(* CODESYS project TP_INF_IND_RENAN_JULIA.project

Project tree, tasks and I/O mapping:
  Device : CODESYS Control Win V3, 3S - Smart Software Solutions GmbH, order no. 305021, version 3.5.11.40
    application Application
      libraries: Standard, * (System)
      task MainTask (cyclic, interval t#10ms, priority 1) calls Main
      task SimulacaoTask (cyclic, interval t#100ms, priority 1) calls SimulacaoProcesso
      program Main [ST]
      program SimulacaoProcesso [ST]
      global variables Variaveis_globais
      function block ControleCarregamento [ST]
      function block ControleDescarregamento [ST]
      function block ManualControl [ST]
      function block gestaoAlarmes [ST]
*)

// Device/Application/Variaveis_globais

VAR_GLOBAL
    // Variáveis de Peso dos Silos
    PESO_SILO1: REAL;
    PESO_SILO2: REAL;
	PESO_MOEGA: REAL;
	CAPACIDADE_SILO : REAL := 2500;
	CAPACIDADE_VAGAO: INT  := 1000;
	CAPACIDADE_ARMAZENAMENTO_SILOS : REAL;
	CAMINHAO_CAPAZ : BOOL;
	INICIAR_CARREGAMENTO : BOOL;
	INICIAR_DESCARREGAMENTO : BOOL;
	VAGAO_POSICIONADO : BOOL;
	PESO_TRANSPORTADOR_ENTRADA : REAL;

    // Indicadores de Nível Alto dos Silos
    NIVEL_ALTO_SILO1: BOOL;
    NIVEL_ALTO_SILO2: BOOL;
    NIVEL_BAIXO_SILO1: BOOL;
	NIVEL_BAIXO_SILO2: BOOL;
    // Posicionamento do Caminhão
    CAMINHAO_POSICIONADO: BOOL;

    // Capacidade do Caminhão
    CAPACIDADE_CAMINHAO: REAL;

    // Comandos para Iniciar Processos
    CMD_INICIAR_DESCARREGAMENTO: BOOL;
    CMD_INICIAR_CARREGAMENTO: BOOL;

    // Estados dos Transportadores
    TRANSPORTADOR_ENTRADA_ON: BOOL;
    TRANSPORTADOR_SAIDA_ON: BOOL;

    // Estados de Ventilação dos Silos
    VENTILACAO_SILO1: BOOL;
    VENTILACAO_SILO2: BOOL;

    // Estado do Alimentador da Moega
    ALIMENTADOR_MOEGA1_ON: BOOL;
	ALIMENTADOR_MOEGA2_ON: BOOL;
	SENSOR_ALIMENTADOR_MOEGA1: BOOL;
	SENSOR_ALIMENTADOR_MOEGA2: BOOL;
    
    // Estados dos Alimentadores de Saída
    ALIMENTADOR_SAIDA_ON: BOOL;
    MOEGA_PESAGEM_ON: BOOL;
    ALIMENTADOR_MOEGA1: BOOL;
    ALIMENTADOR_MOEGA2: BOOL;
	

    // Posição do Desviador de Mangueira
    DESVIADOR_MANGUEIRA_POS: INT;

    // Alarmes
    ALARME_ALIMENTADOR_SAIDA: BOOL;
    ALARME_TRANSPORTADOR_ENTRADA: BOOL;
    ALARME_TRANSPORTADOR_SAIDA: BOOL;
    ALARME_VENTILACAO_SILO1: BOOL;
    ALARME_VENTILACAO_SILO2: BOOL;
	ALARME_CARREGAMENTO: BOOL;
	ALARME_MOEGA: BOOL;
	ALARME_ALIMENTADOR_MOEGA1: BOOL;
	ALARME_ALIMENTADOR_MOEGA2: BOOL;
	ALARME_DESCARREGAMENTO : BOOL;

    // Comandos Manuais
    MANUAL_CMD_TRANSPORTADOR_ENTRADA: BOOL;
    MANUAL_CMD_TRANSPORTADOR_SAIDA: BOOL;
    MANUAL_CMD_VENTILACAO_SILO1: BOOL;
    MANUAL_CMD_VENTILACAO_SILO2: BOOL;
    MANUAL_CMD_ALIMENTADOR_MOEGA: BOOL;

    // Sensores de Posicionamento
    SENSOR_POSICIONAMENTO_VAGAO: BOOL;
    SENSOR_POSICIONAMENTO_CAMINHAO: BOOL;
END_VAR

// Device/Application/Main
PROGRAM Main
VAR
    mode: BOOL; 
    controleDescarregamento: ControleDescarregamento;
    controleCarregamento: ControleCarregamento;
   // simulacaoProcesso: SimulacaoProcesso;
    gestaoAlarmes: GestaoAlarmes;
    manualControl: ManualControl;
    
END_VAR

// Chamar os blocos de controle conforme o modo de operação
IF mode THEN // Modo automático
    controleDescarregamento();
    controleCarregamento();
ELSE // Modo manual
    manualControl();
END_IF

// Simulação e gestão de alarmes
//simulacaoProcesso();
gestaoAlarmes();

END_PROGRAM

// Device/Application/ControleDescarregamento
FUNCTION_BLOCK ControleDescarregamento
VAR
    tempo: TIME := T#0s;
    inicio_descarregamento: TIME;
END_VAR

CAPACIDADE_ARMAZENAMENTO_SILOS := (2400 - PESO_SILO1) + (2400 - PESO_SILO2);


IF (CAPACIDADE_ARMAZENAMENTO_SILOS >= CAPACIDADE_VAGAO) AND (VAGAO_POSICIONADO) THEN
	IF CMD_INICIAR_DESCARREGAMENTO THEN
		IF (NOT VENTILACAO_SILO2) AND (NOT VENTILACAO_SILO1) AND (NOT TRANSPORTADOR_ENTRADA_ON) THEN
          IF (NOT ALARME_TRANSPORTADOR_ENTRADA) AND (NOT ALARME_TRANSPORTADOR_SAIDA) AND (NOT ALARME_VENTILACAO_SILO1) AND (NOT ALARME_VENTILACAO_SILO2) AND (NOT ALARME_ALIMENTADOR_MOEGA1)AND (NOT ALARME_ALIMENTADOR_MOEGA2) AND (NOT ALARME_ALIMENTADOR_SAIDA) AND (NOT ALARME_MOEGA) THEN
		          INICIAR_DESCARREGAMENTO := TRUE;
	      ELSE
		          INICIAR_DESCARREGAMENTO := FALSE;
		          ALARME_DESCARREGAMENTO  := TRUE;
		  END_IF
		END_IF
	END_IF
ELSE
	 INICIAR_DESCARREGAMENTO := FALSE;
     ALARME_DESCARREGAMENTO  := TRUE;
END_IF


IF INICIAR_DESCARREGAMENTO THEN
	
    IF (PESO_SILO1 > PESO_SILO2) OR (PESO_SILO1 = PESO_SILO2 AND DESVIADOR_MANGUEIRA_POS = 2) THEN
        DESVIADOR_MANGUEIRA_POS := 2;
        VENTILACAO_SILO2 := TRUE;
        ALIMENTADOR_MOEGA2_ON := TRUE;
        TRANSPORTADOR_ENTRADA_ON := TRUE;
        inicio_descarregamento := TIME();

        IF (NIVEL_ALTO_SILO2) THEN
            ALIMENTADOR_MOEGA2_ON := FALSE;
            TRANSPORTADOR_ENTRADA_ON := FALSE;
            VENTILACAO_SILO2 := FALSE;
            DESVIADOR_MANGUEIRA_POS := 1;
        END_IF
		
    ELSE
        DESVIADOR_MANGUEIRA_POS := 1;
        VENTILACAO_SILO1 := TRUE;
        ALIMENTADOR_MOEGA1_ON := TRUE;
        TRANSPORTADOR_ENTRADA_ON := TRUE;
        inicio_descarregamento := TIME();

        IF (NIVEL_ALTO_SILO1) THEN
            ALIMENTADOR_MOEGA1_ON := FALSE;
            TRANSPORTADOR_ENTRADA_ON := FALSE;
            VENTILACAO_SILO1 := FALSE;
            DESVIADOR_MANGUEIRA_POS := 2;
        END_IF

    END_IF
END_IF

IF PESO_TRANSPORTADOR_ENTRADA = 0 THEN

            tempo := TIME() - inicio_descarregamento;
            IF (tempo >= T#2S) THEN
               TRANSPORTADOR_ENTRADA_ON := FALSE;
            END_IF
            IF (tempo >= T#5S) THEN
               VENTILACAO_SILO1 := FALSE;
			   VENTILACAO_SILO2 := FALSE;
            END_IF
		
END_IF

END_FUNCTION_BLOCK

// Device/Application/ControleCarregamento
FUNCTION_BLOCK ControleCarregamento
VAR
    tempo: TIME := T#0s;
    inicio_carregamento: TIME;
    INICIAR_CARREGAMENTO: BOOL := FALSE;
    ALARME_CARREGAMENTO: BOOL := FALSE;
    CAPACIDADE_CAMINHAO: REAL := 0.0; // Inicialização para um valor padrão
    CAMINHAO_CAPAZ: BOOL := FALSE;
    CAMINHAO_POSICIONADO: BOOL := FALSE;
    PESO_SILO1: REAL := 0.0; // Inicialização para um valor padrão
    PESO_SILO2: REAL := 0.0; // Inicialização para um valor padrão
    VENTILACAO_SILO1: BOOL := FALSE;
    VENTILACAO_SILO2: BOOL := FALSE;
    TRANSPORTADOR_ENTRADA_ON: BOOL := FALSE;
    SENSOR_ALIMENTADOR_MOEGA1: BOOL := FALSE;
    SENSOR_ALIMENTADOR_MOEGA2: BOOL := FALSE;
    ALIMENTADOR_SAIDA_ON: BOOL := FALSE;
    TRANSPORTADOR_SAIDA_ON: BOOL := FALSE;
    MOEGA_PESAGEM_ON: BOOL := FALSE;
    ALIMENTADOR_MOEGA1_ON: BOOL := FALSE;
    ALIMENTADOR_MOEGA2_ON: BOOL := FALSE;
    ALARME_TRANSPORTADOR_ENTRADA: BOOL := FALSE;
    ALARME_TRANSPORTADOR_SAIDA: BOOL := FALSE;
    ALARME_VENTILACAO_SILO1: BOOL := FALSE;
    ALARME_VENTILACAO_SILO2: BOOL := FALSE;
    ALARME_ALIMENTADOR_MOEGA1: BOOL := FALSE;
    ALARME_ALIMENTADOR_MOEGA2: BOOL := FALSE;
    ALARME_ALIMENTADOR_SAIDA: BOOL := FALSE;
    ALARME_MOEGA: BOOL := FALSE;
END_VAR

IF (CAPACIDADE_CAMINHAO >= 200) AND (CAPACIDADE_CAMINHAO <= 800)THEN
	CAMINHAO_CAPAZ := TRUE;
ELSE
	CAMINHAO_CAPAZ := FALSE;
END_IF

IF CAMINHAO_CAPAZ AND CAMINHAO_POSICIONADO THEN //VERIFICA SE O CAMINHAO TEM CAPACIDADE E ESTÁ POSICIONADO
	IF CMD_INICIAR_CARREGAMENTO THEN            //SE RECEBER COMANDO DO OPERADOR  
  		 IF (NOT VENTILACAO_SILO2) AND (NOT VENTILACAO_SILO1) AND (NOT TRANSPORTADOR_ENTRADA_ON) AND (NOT SENSOR_ALIMENTADOR_MOEGA1) AND (NOT SENSOR_ALIMENTADOR_MOEGA2) AND (NOT ALIMENTADOR_SAIDA_ON) AND (NOT TRANSPORTADOR_SAIDA_ON) AND (NOT MOEGA_PESAGEM_ON) AND (NOT ALIMENTADOR_MOEGA1) AND (NOT ALIMENTADOR_MOEGA2) THEN
			 IF (NOT ALARME_TRANSPORTADOR_ENTRADA) AND (NOT ALARME_TRANSPORTADOR_SAIDA) AND (NOT ALARME_VENTILACAO_SILO1) AND (NOT ALARME_VENTILACAO_SILO2) AND (NOT ALARME_ALIMENTADOR_MOEGA1)AND (NOT ALARME_ALIMENTADOR_MOEGA2) AND (NOT ALARME_ALIMENTADOR_SAIDA) AND (NOT ALARME_MOEGA) THEN
				 IF (PESO_SILO1 - 100) + (PESO_SILO2 - 100) >= CAPACIDADE_CAMINHAO THEN
                    INICIAR_CARREGAMENTO := TRUE;
                ELSE
                    ALARME_CARREGAMENTO := TRUE;
					INICIAR_CARREGAMENTO := FALSE;
                END_IF
            END_IF
        END_IF
    END_IF
END_IF

IF INICIAR_CARREGAMENTO THEN
    IF (PESO_SILO1 >= PESO_SILO2) THEN
        VENTILACAO_SILO1 := TRUE;
        ALIMENTADOR_SAIDA_ON := TRUE;
        TRANSPORTADOR_SAIDA_ON := TRUE;
        MOEGA_PESAGEM_ON := TRUE;
        ALIMENTADOR_MOEGA1 := TRUE;

        // Esperar até que a pesagem atinja o valor informado
        IF (PESO_MOEGA >= CAPACIDADE_CAMINHAO) THEN
            ALIMENTADOR_MOEGA1 := FALSE;
            VENTILACAO_SILO1 := FALSE;
            ALIMENTADOR_SAIDA_ON := FALSE;
            TRANSPORTADOR_SAIDA_ON := FALSE;
            MOEGA_PESAGEM_ON := FALSE;
			INICIAR_CARREGAMENTO := FALSE;
        ELSE
            IF (NIVEL_BAIXO_SILO1) THEN
                ALIMENTADOR_MOEGA1 := FALSE;
                VENTILACAO_SILO1 := FALSE;
                ALIMENTADOR_SAIDA_ON := FALSE;
                TRANSPORTADOR_SAIDA_ON := FALSE;
                MOEGA_PESAGEM_ON := FALSE;

                ALIMENTADOR_MOEGA2 := TRUE;
                VENTILACAO_SILO2 := TRUE;
                ALIMENTADOR_SAIDA_ON := TRUE;
                TRANSPORTADOR_SAIDA_ON := TRUE;
                MOEGA_PESAGEM_ON := TRUE;

                IF (PESO_MOEGA >= CAPACIDADE_CAMINHAO) THEN
                    ALIMENTADOR_MOEGA2 := FALSE;
					INICIAR_CARREGAMENTO := FALSE;
                END_IF
            END_IF
        END_IF

        // Controle de tempo e desativação dos equipamentos
        inicio_carregamento := TIME();
        IF (TIME() - inicio_carregamento >= T#1S) THEN
            MOEGA_PESAGEM_ON := FALSE;
        END_IF
        IF (TIME() - inicio_carregamento >= T#2S) THEN
            TRANSPORTADOR_SAIDA_ON := FALSE;
        END_IF
        IF (TIME() - inicio_carregamento >= T#3S) THEN
            ALIMENTADOR_SAIDA_ON := FALSE;
        END_IF
        IF (TIME() - inicio_carregamento >= T#5S) THEN
            VENTILACAO_SILO1 := FALSE;
        END_IF

    ELSE
        VENTILACAO_SILO2 := TRUE;
        ALIMENTADOR_SAIDA_ON := TRUE;
        TRANSPORTADOR_SAIDA_ON := TRUE;
        MOEGA_PESAGEM_ON := TRUE;
        ALIMENTADOR_MOEGA2 := TRUE;

        // Esperar até que a pesagem atinja o valor informado
        IF (PESO_MOEGA >= CAPACIDADE_CAMINHAO) THEN
            ALIMENTADOR_MOEGA2 := FALSE;
            VENTILACAO_SILO2 := FALSE;
            ALIMENTADOR_SAIDA_ON := FALSE;
            TRANSPORTADOR_SAIDA_ON := FALSE;
            MOEGA_PESAGEM_ON := FALSE;
			INICIAR_CARREGAMENTO := FALSE;
        ELSE
            IF (NIVEL_BAIXO_SILO2) THEN
                ALIMENTADOR_MOEGA2 := FALSE;
                VENTILACAO_SILO2 := FALSE;
                ALIMENTADOR_SAIDA_ON := FALSE;
                TRANSPORTADOR_SAIDA_ON := FALSE;
                MOEGA_PESAGEM_ON := FALSE;

                ALIMENTADOR_MOEGA1 := TRUE;
                VENTILACAO_SILO1 := TRUE;
                ALIMENTADOR_SAIDA_ON := TRUE;
                TRANSPORTADOR_SAIDA_ON := TRUE;
                MOEGA_PESAGEM_ON := TRUE;

                IF (PESO_MOEGA >= CAPACIDADE_CAMINHAO) THEN
                    ALIMENTADOR_MOEGA1 := FALSE;
					INICIAR_CARREGAMENTO := FALSE;
                END_IF
            END_IF
        END_IF

        // Controle de tempo e desativação dos equipamentos
        inicio_carregamento := TIME();
        IF (TIME() - inicio_carregamento >= T#1S) THEN
            MOEGA_PESAGEM_ON := FALSE;
        END_IF
        IF (TIME() - inicio_carregamento >= T#2S) THEN
            TRANSPORTADOR_SAIDA_ON := FALSE;
        END_IF
        IF (TIME() - inicio_carregamento >= T#3S) THEN
            ALIMENTADOR_SAIDA_ON := FALSE;
        END_IF
        IF (TIME() - inicio_carregamento >= T#5S) THEN
            VENTILACAO_SILO2 := FALSE;
        END_IF
    END_IF
END_IF

END_FUNCTION_BLOCK

// Device/Application/ManualControl
FUNCTION_BLOCK ManualControl
VAR_INPUT
    MANUAL_CMD_TRANSPORTADOR_ENTRADA: BOOL;
    MANUAL_CMD_TRANSPORTADOR_SAIDA: BOOL;
    MANUAL_CMD_VENTILACAO_SILO1: BOOL;
    MANUAL_CMD_VENTILACAO_SILO2: BOOL;
    MANUAL_CMD_ALIMENTADOR_MOEGA: BOOL;
    
END_VAR

VAR_OUTPUT
    TRANSPORTADOR_ENTRADA_ON: BOOL;
    TRANSPORTADOR_SAIDA_ON: BOOL;
    VENTILACAO_SILO1: BOOL;
    VENTILACAO_SILO2: BOOL;
    ALIMENTADOR_MOEGA_ON: BOOL;
    
END_VAR


TRANSPORTADOR_ENTRADA_ON := MANUAL_CMD_TRANSPORTADOR_ENTRADA;
TRANSPORTADOR_SAIDA_ON := MANUAL_CMD_TRANSPORTADOR_SAIDA;
VENTILACAO_SILO1 := MANUAL_CMD_VENTILACAO_SILO1;
VENTILACAO_SILO2 := MANUAL_CMD_VENTILACAO_SILO2;
ALIMENTADOR_MOEGA_ON := MANUAL_CMD_ALIMENTADOR_MOEGA;

END_FUNCTION_BLOCK

// Device/Application/SimulacaoProcesso
PROGRAM SimulacaoProcesso
VAR_INPUT
    TRANSPORTADOR_ENTRADA_ON: BOOL;
    TRANSPORTADOR_SAIDA_ON: BOOL;
    VENTILACAO_SILO1: BOOL;
    VENTILACAO_SILO2: BOOL;
    ALIMENTADOR_MOEGA1_ON: BOOL;
    ALIMENTADOR_MOEGA2_ON: BOOL;
    CAMINHAO_POSICIONADO: BOOL;
    VAGAO_POSICIONADO: BOOL;
END_VAR

VAR_OUTPUT
    PESO_SILO1: REAL;
    PESO_SILO2: REAL;
    PESO_MOEGA: REAL;
    SENSOR_GRAO_ALIMENTADOR_MOEGA1: BOOL;
    SENSOR_GRAO_ALIMENTADOR_MOEGA2: BOOL;
    NIVEL_ALTO_SILO1: BOOL;
    NIVEL_ALTO_SILO2: BOOL;
    NIVEL_BAIXO_SILO1: BOOL;
    NIVEL_BAIXO_SILO2: BOOL;
    PESO_TRANSPORTADOR_ENTRADA: REAL;
    PESO_TRANSPORTADOR_SAIDA: REAL;
END_VAR

VAR
    taxa_transferencia: REAL := 50.0; // Taxa de transferência dos transportadores (kg/s)
    tempo_atual: TIME;
    tempo_anterior: TIME := T#0s;
    delta_t: REAL;
END_VAR

// Calcular delta_t
tempo_atual := TIME();
delta_t := TIME_TO_REAL(tempo_atual - tempo_anterior) / 1000.0; // Converter TIME para segundos

// Inicializar variáveis de saída
PESO_TRANSPORTADOR_ENTRADA := 0.0;
PESO_TRANSPORTADOR_SAIDA := 0.0;

// Simular o comportamento dos silos e transportadores
IF TRANSPORTADOR_ENTRADA_ON THEN
    PESO_TRANSPORTADOR_ENTRADA := taxa_transferencia * delta_t;
    IF ALIMENTADOR_MOEGA1_ON THEN
        PESO_SILO1 := PESO_SILO1 + PESO_TRANSPORTADOR_ENTRADA;
        PESO_MOEGA := PESO_MOEGA - PESO_TRANSPORTADOR_ENTRADA;
    ELSIF ALIMENTADOR_MOEGA2_ON THEN
        PESO_SILO2 := PESO_SILO2 + PESO_TRANSPORTADOR_ENTRADA;
        PESO_MOEGA := PESO_MOEGA - PESO_TRANSPORTADOR_ENTRADA;
    END_IF
END_IF

IF TRANSPORTADOR_SAIDA_ON THEN
    PESO_TRANSPORTADOR_SAIDA := taxa_transferencia * delta_t;
    IF ALIMENTADOR_MOEGA1_ON THEN
        PESO_MOEGA := PESO_MOEGA + PESO_TRANSPORTADOR_SAIDA;
        PESO_SILO1 := PESO_SILO1 - PESO_TRANSPORTADOR_SAIDA;
    ELSIF ALIMENTADOR_MOEGA2_ON THEN
        PESO_MOEGA := PESO_MOEGA + PESO_TRANSPORTADOR_SAIDA;
        PESO_SILO2 := PESO_SILO2 - PESO_TRANSPORTADOR_SAIDA;
    END_IF
END_IF

// Atualizar sensores de grãos
SENSOR_GRAO_ALIMENTADOR_MOEGA1 := (PESO_SILO1 > 0);
SENSOR_GRAO_ALIMENTADOR_MOEGA2 := (PESO_SILO2 > 0);

// Verificar níveis altos e baixos dos silos
NIVEL_ALTO_SILO1 := (PESO_SILO1 >= 2400);
NIVEL_ALTO_SILO2 := (PESO_SILO2 >= 2400);
NIVEL_BAIXO_SILO1 := (PESO_SILO1 <= 100);
NIVEL_BAIXO_SILO2 := (PESO_SILO2 <= 100);

// Atualizar o tempo anterior
tempo_anterior := tempo_atual;

END_PROGRAM

// Device/Application/gestaoAlarmes
FUNCTION_BLOCK GestaoAlarmes
VAR_INPUT
    TRANSPORTADOR_ENTRADA_ON: BOOL;
    TRANSPORTADOR_SAIDA_ON: BOOL;
    VENTILACAO_SILO1: BOOL;
    VENTILACAO_SILO2: BOOL;
    ALIMENTADOR_MOEGA1_ON: BOOL;
    ALIMENTADOR_MOEGA2_ON: BOOL;
    PESO_TRANSPORTADOR_ENTRADA: REAL;
    PESO_TRANSPORTADOR_SAIDA: REAL;
    PESO_MOEGA: REAL;
    SENSOR_GRAO_ALIMENTADOR_MOEGA1: BOOL;
    SENSOR_GRAO_ALIMENTADOR_MOEGA2: BOOL;
    CAMINHAO_POSICIONADO: BOOL;
    PESO_SILO1: REAL;
    PESO_SILO2: REAL;
END_VAR

VAR_OUTPUT
    ALARME_TRANSPORTADOR_ENTRADA: BOOL;
    ALARME_TRANSPORTADOR_SAIDA: BOOL;
    ALARME_VENTILACAO_SILO1: BOOL;
    ALARME_VENTILACAO_SILO2: BOOL;
    ALARME_ALIMENTADOR_MOEGA1: BOOL;
    ALARME_ALIMENTADOR_MOEGA2: BOOL;
    ALARME_ALIMENTADOR_SAIDA: BOOL;
    ALARME_MOEGA: BOOL;
    ALARME_NIVEL_BAIXO_SILO1: BOOL;
    ALARME_NIVEL_BAIXO_SILO2: BOOL;
    ALARME_NIVEL_ALTO_SILO1: BOOL;
    ALARME_NIVEL_ALTO_SILO2: BOOL;
END_VAR

VAR
    tempo_transportador_entrada: TIME;
    tempo_transportador_saida: TIME;
    tempo_alimentador_moega1: TIME;
    tempo_alimentador_moega2: TIME;
    inicio_transportador_entrada: TIME;
    inicio_transportador_saida: TIME;
    inicio_alimentador_moega1: TIME;
    inicio_alimentador_moega2: TIME;
END_VAR

IF NOT TRANSPORTADOR_ENTRADA_ON THEN
    inicio_transportador_entrada := TIME();
    ALARME_TRANSPORTADOR_ENTRADA := FALSE;
ELSE
    tempo_transportador_entrada := TIME() - inicio_transportador_entrada;
    IF (tempo_transportador_entrada >= T#5S) AND (PESO_TRANSPORTADOR_ENTRADA = 0) THEN
        ALARME_TRANSPORTADOR_ENTRADA := TRUE;
    END_IF
END_IF

IF NOT TRANSPORTADOR_SAIDA_ON THEN
    inicio_transportador_saida := TIME();
    ALARME_TRANSPORTADOR_SAIDA := FALSE;
ELSE
    tempo_transportador_saida := TIME() - inicio_transportador_saida;
    IF (tempo_transportador_saida >= T#5S) AND (PESO_TRANSPORTADOR_SAIDA = 0) THEN
        ALARME_TRANSPORTADOR_SAIDA := TRUE;
    END_IF
    IF (TRANSPORTADOR_SAIDA_ON) AND (NOT ALIMENTADOR_SAIDA_ON) THEN
        ALARME_TRANSPORTADOR_SAIDA := TRUE;
    END_IF
END_IF

IF (ALIMENTADOR_SAIDA_ON AND NOT CAMINHAO_POSICIONADO) THEN
   ALARME_ALIMENTADOR_SAIDA := TRUE;
ELSE
   ALARME_ALIMENTADOR_SAIDA := FALSE;
END_IF

IF (NOT TRANSPORTADOR_SAIDA_ON) AND (PESO_MOEGA > 0) THEN
    ALARME_MOEGA := TRUE;
ELSE
    ALARME_MOEGA := FALSE;
END_IF

IF ALIMENTADOR_MOEGA1_ON THEN
    IF NOT SENSOR_ALIMENTADOR_MOEGA1 THEN
        inicio_alimentador_moega1 := TIME();
        tempo_alimentador_moega1 := TIME() - inicio_alimentador_moega1;
        IF tempo_alimentador_moega1 >= T#5S THEN
            ALARME_ALIMENTADOR_MOEGA1 := TRUE;
        END_IF
    ELSE
        ALARME_ALIMENTADOR_MOEGA1 := FALSE;
    END_IF
ELSE
    inicio_alimentador_moega1 := TIME();
END_IF

IF ALIMENTADOR_MOEGA2_ON THEN
    IF NOT SENSOR_ALIMENTADOR_MOEGA2 THEN
        inicio_alimentador_moega2 := TIME();
        tempo_alimentador_moega2 := TIME() - inicio_alimentador_moega2;
        IF tempo_alimentador_moega2 >= T#5S THEN
            ALARME_ALIMENTADOR_MOEGA2 := TRUE;
        END_IF
    ELSE
        ALARME_ALIMENTADOR_MOEGA2 := FALSE;
    END_IF
ELSE
    inicio_alimentador_moega2 := TIME();
END_IF

IF PESO_SILO1 < 100 THEN
    NIVEL_BAIXO_SILO1 := TRUE;
ELSE
    NIVEL_BAIXO_SILO1 := FALSE;
END_IF

IF PESO_SILO2 < 100 THEN
    NIVEL_BAIXO_SILO2 := TRUE;
ELSE
    NIVEL_BAIXO_SILO2 := FALSE;
END_IF

IF PESO_SILO1 > 2400 THEN
    NIVEL_ALTO_SILO1 := TRUE;
ELSE
    NIVEL_ALTO_SILO1 := FALSE;
END_IF

IF PESO_SILO2 > 2400 THEN
    NIVEL_ALTO_SILO2 := TRUE;
ELSE
    NIVEL_ALTO_SILO2 := FALSE;
END_IF

END_FUNCTION_BLOCK
